// Mitsubishi GX Works2 project: 0907QR   PLC: Q03UDV

PROGRAM MAIN
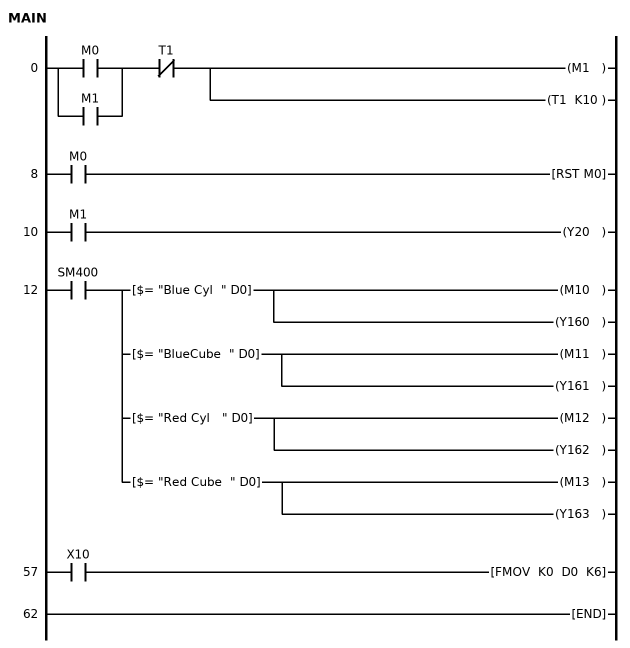
0     LD      M0
      OR      M1
      ANI     T1
      OUT     M1
      OUT     T1 K10
8     LD      M0
      RST     M0
10    LD      M1
      OUT     Y20
12    LD      SM400
      MPS
      AND$=   "Blue Cyl  " D0
      OUT     M10
      OUT     Y160
      MRD
      AND$=   "BlueCube  " D0
      OUT     M11
      OUT     Y161
      MRD
      AND$=   "Red Cyl   " D0
      OUT     M12
      OUT     Y162
      MPP
      AND$=   "Red Cube  " D0
      OUT     M13
      OUT     Y163
57    LD      X10
      FMOV    K0 D0 K6
62    END
END_PROGRAM

PROGRAM MAIN1
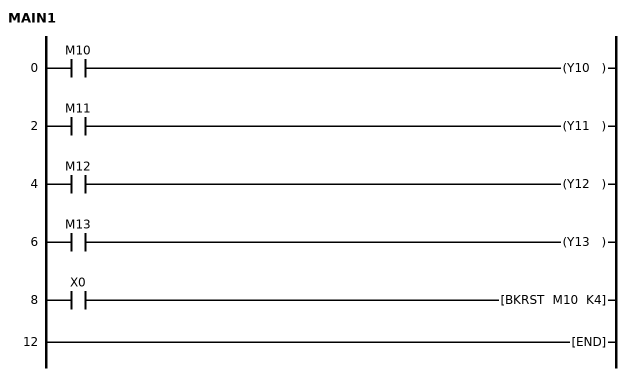
0     LD      M10
      OUT     Y10
2     LD      M11
      OUT     Y11
4     LD      M12
      OUT     Y12
6     LD      M13
      OUT     Y13
8     LD      X0
      BKRST   M10 K4
12    END
END_PROGRAM
